(*
An abstract representation of a system state, providing the foundation for implementing state-specific behavior.  
Manages its owner entity and supports state transitions within the system.  
Offers default behavior for state lifecycle methods, allowing programmers to override only the relevant parts.
*)
FUNCTION_BLOCK ABSTRACT State IMPLEMENTS I_StateInternal, I_State
VAR
	{attribute 'hide'}
	_tag						: Tag('');
	{attribute 'hide'}
	_bInQueue					: BOOL;
	{attribute 'hide'}
	_iOwner						: I_Entity;
END_VAR

PROPERTY INTERNAL FINAL _AsIState : I_State
GET
_AsIState := THIS^;
END_GET
END_PROPERTY

PROPERTY INTERNAL FINAL _AsIStateInternal : I_StateInternal
GET
_AsIStateInternal := THIS^;
END_GET
END_PROPERTY

PROPERTY INTERNAL FINAL _InQueue : BOOL
GET
_InQueue := _bInQueue;
END_GET
SET
_bInQueue := _InQueue;
END_SET
END_PROPERTY

(*
Determines whether the state can be activated.  
Returns `TRUE` by default but can be overridden for specific activation conditions.
*)
METHOD CanActivate : BOOL
CanActivate := TRUE;
END_METHOD

(*
Determines whether the state can be deactivated.  
Returns `TRUE` by default but can be overridden for specific deactivation conditions.
*)
METHOD CanDeactivate : BOOL
CanDeactivate := TRUE;
END_METHOD

//FB_Init is always available implicitly and it is used primarily for initialization.
//The return value is not evaluated. For a specific influence, you can also declare the
//methods explicitly and provide additional code there with the standard initialization
//code. You can evaluate the return value.
METHOD FB_Init: BOOL
VAR_INPUT
    bInitRetains: BOOL; // TRUE: the retain variables are initialized (reset warm / reset cold)
    bInCopyCode: BOOL;  // TRUE: the instance will be copied to the copy code afterward (online change)
	
	iEntity		: I_Entity;
END_VAR
VAR
	_nResult	: Result;
END_VAR
IF iEntity = 0 THEN
	DebugMsg(THIS^, 'iEntity = 0!');
END_IF

_iOwner := iEntity;;

IF IsErr(_RegComp(iEntity, THIS^), nOut => _nResult) THEN
	DebugMsg(THIS^, Tc2_Standard.CONCAT('Failed with code: ', TO_STRING(_nResult)));
	DebugMsg(THIS^, 'Could not be added!');
END_IF
END_METHOD

(*
Executed when the state is entered.  
Provides a hook for defining state-specific behavior to be performed during the transition into this state.
*)
METHOD OnEntry
END_METHOD

(*
Executed during the state's operation.  
Used to define state-specific logic that runs while the state is active.
*)
METHOD OnExecute
END_METHOD

(*
Executed when the state transitions to another state.  
Provides a hook for defining cleanup or transition-specific behavior.
*)
METHOD OnExit
END_METHOD

(*
Returns the entity that owns this state.
*)
PROPERTY FINAL Owner : I_Entity
GET
Owner := _iOwner;
END_GET
END_PROPERTY

(*
Provides access to the `I_Tag` associated with the state.
*)
PROPERTY FINAL Tag : I_Tag
GET
Tag := _tag;
END_GET
END_PROPERTY

END_FUNCTION_BLOCK

(* stored: Version 1.1.0.1
   POU State: Id {a3b28716-f684-494e-889b-84fe1781ad45}, SpecialFunc None
   Folder _: Id {b2082cde-a72a-48d1-bf2b-bfe685440ba0}
   Folder Can: Id {012b303c-ee19-4d59-a8c5-29d7ee56e39c}
   Folder On: Id {5034b126-7af1-4e3e-aa65-10d454bc5f51}
   Property _AsIState: Id {ae988e03-7493-46d9-85de-be6948de1d8e}
   Get Get: Id {4c9d6b0d-006b-455b-828d-2ce5937584f8}
   Property _AsIStateInternal: Id {4fe75cff-cf53-4cef-a5a6-8ca77becdd1c}
   Get Get: Id {d8d590d5-9436-40ea-add0-78eaf9a46d23}
   Property _InQueue: Id {7211bf2e-3f54-4127-8169-2b1f66f2bb49}
   Get Get: Id {f6028f30-7546-40bc-a7f1-f2d9bdc4c404}
   Set Set: Id {2b151194-8b26-4b93-a27d-8d175bcf9d22}
   Method CanActivate: Id {71c49a83-838e-4656-9fc2-ce8957b8e198}
   Method CanDeactivate: Id {d9ac8857-b429-40a0-ae64-2f200213bb6e}
   Method FB_init: Id {2842d681-0b8d-4523-860b-e4e2b7025ae0}
   Method OnEntry: Id {233f0cb7-a018-4a8e-a04c-cd20357f448f}
   Method OnExecute: Id {aabb82b9-2f5d-4e99-b353-6c10e3d6ce3d}
   Method OnExit: Id {25d7c89a-22df-4af1-9c2c-e2be2f3e48a9}
   Property Owner: Id {32b502a4-ba25-4a78-8e46-5a8b31e2a3e9}
   Get Get: Id {98a99666-df4c-40b9-abec-3c308e3cdead}
   Property Tag: Id {0bbeba40-ec6e-4b6d-a33f-9c84eca9c89e}
   Get Get: Id {c1b1ddfd-4e01-4e44-9d81-1a59ffd92985} *)
